(* Copyright 2017 Cimpress

Licensed under the Apache License, Version 2.0 (the "License");
you may not use this file except in compliance with the License.
You may obtain a copy of the License at

http://www.apache.org/licenses/LICENSE-2.0

Unless required by applicable law or agreed to in writing, software
distributed under the License is distributed on an "AS IS" BASIS,
WITHOUT WARRANTIES OR CONDITIONS OF ANY KIND, either express or implied.
See the License for the specific language governing permissions and
limitations under the License. *)

TYPE T_FileLc_SysCfg :
STRUCT
	uinMaxNbrOfLogFiles : UINT; (*Maximale Anzahl Log-Files*)
	udiTimeCheckMaxFileNr :UDINT; // [ms] time until check if more then max number of files exist in folder -> delete oldest
	uinNewFileOnRestart : UINT; (*Nach Steuerungsneustart neues File anlegen, wenn Wert > 0*)
	udiMaxTimeWriteToFile : UDINT; (*Maximale Zeit zwischen zwei File - Schreibzyklen*)
	bolUseLocalTimeStamp : BOOL; // define if using local time or UTC
	strLogFileNameExt : STRING[FileLc.cFILENAME_LENGTH]; (*Extension des Logfiles*)
	strLogFileNamePraeFix : STRING[FileLc.cFILENAME_LENGTH]; (*Präfix des Logfiles*)
	strLogPath : STRING[FileLc.cFILENAME_LENGTH]; (*Verzeichnis in welchem die Logfiles angelegt werden*)
	strLogNetId : STRING(23); // to access foreign system drives where TinCat has to be installed!!! Is a string containing the AMS network identifier of the target device to which the ADS command is directed.
	udiQueueLen : UDINT; (*Queue Länge der BaseLog - Queue*)
	udiMaxFileSize : UDINT; (*Maximale Dateigrösse eines Logfiles*)
	udiMaxEntriesInFile : UDINT; (*Maximale Anzahl Einträge in einem Logfile*)
END_STRUCT
END_TYPE

(* stored: Version 1.1.0.1, ProductVersion 3.1.4019.2
   DUT T_FileLc_SysCfg: Id {335d876a-53b4-41b4-b6b0-9197b46aea41} *)
